INTERFACE IComparable EXTENDS IObject

METHOD CompareTo : COMPARISION_RESULT
VAR_INPUT
	object : IObject;
END_VAR
END_METHOD

END_INTERFACE

(* stored: Version 1.1.0.1
   Itf IComparable: Id {b5be0f65-c977-4099-b0bd-3df380b858fb}
   Method CompareTo: Id {e44d871a-9fad-4f68-9d05-06910fe95348} *)
